// working states for FB_ReadHddUsage
{attribute 'qualified_only'}
{attribute 'strict'}
TYPE E_ReadHddUsageStates:
(
  Idle     := 0,
  Letter   := 1,
  Total    := 2,
  Remaining:= 3
);
END_TYPE

(* stored: Version 1.1.0.1, ProductVersion 3.1.4024.4
   DUT E_ReadHddUsageStates: Id {09d6a3e2-e725-4be2-94d7-77284883738a} *)
